GLOBALCONSTANTS CommunicationPartners (* Global constants *)
  (* Standard: 61499-1 *)
  (* Version 1.0, 2025-09-06, franz *)
  PACKAGE isobus;
  VAR_GLOBAL CONSTANT
    GLOBAL : isobus::CF_INFO_T := (s16Handle := BYTE_TO_INT(ADDRESS::GLOBAL_A));
  END_VAR
END_GLOBALCONSTANTS
